SUBAPPLICATION Uebung_009a (* RampLimitFS *)
  (* Standard: 61499-2; Description: Copyright (c) 2023 Meisterschulen am Ostbahnhof This program and the accompanying materials are made available under the terms of the Eclipse Public License 2.0 which is available at https://www.eclipse.org/legal/epl-2.0/ SPDX-License-Identifier: EPL-2.0 *)
  (* Version 1.0, 2023-10-23, Franz Höpfinger, Meisterschulen am Ostbahnhof *)
  IMPORT Uebungen::const::UT::DefaultPool::OutputNumber_N1;
  IMPORT logiBUS::io::DI::logiBUS_DI::Input_I1;
  IMPORT logiBUS::io::DI::logiBUS_DI::Input_I2;
  IMPORT logiBUS::io::DI::logiBUS_DI::Input_I3;
  IMPORT logiBUS::io::DI::logiBUS_DI::Input_I4;
  IMPORT logiBUS::io::DI::logiBUS_DI_Events::BUTTON_LONG_PRESS_START;
  IMPORT logiBUS::io::DI::logiBUS_DI_Events::BUTTON_SINGLE_CLICK;
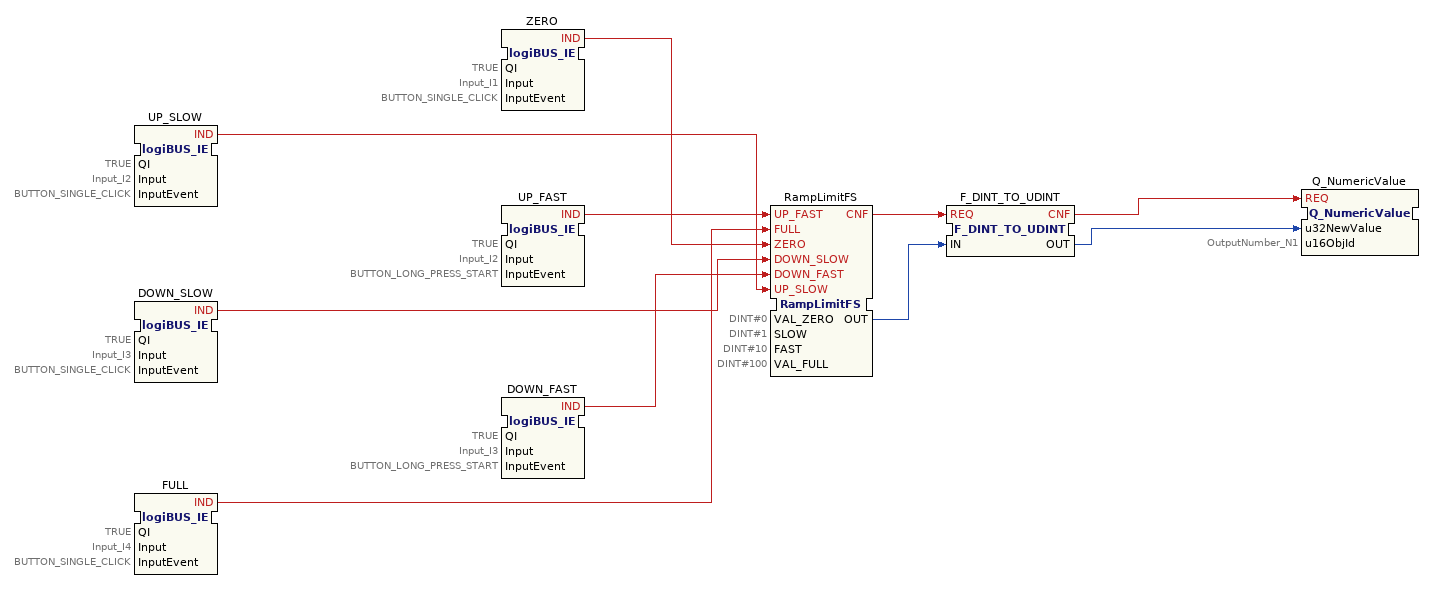
  FBS
    Q_NumericValue : isobus::ut::Q_NumericValue(u16ObjId := OutputNumber_N1);
    UP_FAST : logiBUS::io::DI::logiBUS_IE(QI := TRUE, Input := Input_I2, InputEvent := BUTTON_LONG_PRESS_START);
    DOWN_SLOW : logiBUS::io::DI::logiBUS_IE(QI := TRUE, Input := Input_I3, InputEvent := BUTTON_SINGLE_CLICK);
    F_DINT_TO_UDINT : iec61131::conversion::F_DINT_TO_UDINT;
    ZERO : logiBUS::io::DI::logiBUS_IE(QI := TRUE, Input := Input_I1, InputEvent := BUTTON_SINGLE_CLICK);
    DOWN_FAST : logiBUS::io::DI::logiBUS_IE(QI := TRUE, Input := Input_I3, InputEvent := BUTTON_LONG_PRESS_START);
    UP_SLOW : logiBUS::io::DI::logiBUS_IE(QI := TRUE, Input := Input_I2, InputEvent := BUTTON_SINGLE_CLICK);
    RampLimitFS : eclipse4diac::signalprocessing::RampLimitFS(VAL_ZERO := DINT#0, SLOW := DINT#1, FAST := DINT#10, VAL_FULL := DINT#100);
    FULL : logiBUS::io::DI::logiBUS_IE(QI := TRUE, Input := Input_I4, InputEvent := BUTTON_SINGLE_CLICK);
  END_FBS
  EVENT_CONNECTIONS
    UP_FAST.IND TO RampLimitFS.UP_FAST;
    FULL.IND TO RampLimitFS.FULL;
    RampLimitFS.CNF TO F_DINT_TO_UDINT.REQ;
    ZERO.IND TO RampLimitFS.ZERO;
    DOWN_SLOW.IND TO RampLimitFS.DOWN_SLOW;
    DOWN_FAST.IND TO RampLimitFS.DOWN_FAST;
    UP_SLOW.IND TO RampLimitFS.UP_SLOW;
    F_DINT_TO_UDINT.CNF TO Q_NumericValue.REQ;
  END_CONNECTIONS
  DATA_CONNECTIONS
    RampLimitFS.OUT TO F_DINT_TO_UDINT.IN;
    F_DINT_TO_UDINT.OUT TO Q_NumericValue.u32NewValue;
  END_CONNECTIONS
END_SUBAPPLICATION
